PROGRAM YAG_LimitSwitched

VAR
	
    axisYAG: AXIS_REF;
    fbAxisPowerYAG: MC_Power;
       
	bEnable: BOOL := TRUE;
    fOverride: LREAL := 100;
    		
	biLimFwd_YAG AT %I*: BOOL;
	biLimBwd_YAG AT %I*: BOOL;

	fbtest: FB_TEST;
	I_moter_Yag AT %I*: UINT;
	
END_VAR

fbtest(
	axis:=axisYAG , 
	fTargetVelocity:=0.5 , 
	fStartPosition:= 0, 
	fEndPosition:= 41, 
	nDivisions:= 20 , 
	fbAxisPower:= fbAxisPowerYAG );
fbAxisPowerYAG(
    Axis:= axisYAG,
    Enable:= bEnable,
    Enable_Positive:= biLimFwd_YAG, // TRUE, //
    Enable_Negative:= biLimBwd_YAG, // TRUE, //
    Override:= fOverride,
    BufferMode:= ,
    Options:= ,
    Status=> ,
    Busy=> ,
    Active=> ,
    Error=> ,
    ErrorID=> );

END_PROGRAM

(* stored: Version 1.1.0.1, ProductVersion 3.1.4024.4
   POU YAG_LimitSwitched: Id {926e5d18-980c-4bc0-baa3-64e27920106e}, SpecialFunc None *)
